{attribute addProperty BoxType "EK1122-0000-0018"}
{attribute addProperty Id "Beckhoff_EL73xxsub_EK1100EK1100_179A0949162"}
{attribute addProperty CRC "4226893576"}
{attribute addProperty SizeInBites "16"}
{attribute addProperty SizeInBytes "2"}
TYPE Beckhoff_EL73xxEK1122_FBF14708 EXTENDS EK1122_179A0949 :
STRUCT
	{attribute addProperty Name "Beckhoff_EL73xxsub_EK1100"}
	Beckhoff_EL73xxsub_EK1100 : EK1100_179A0949;
END_STRUCT
END_TYPE

(* stored: Version 1.2.0.0, ProductVersion 3.1.4024.9
   DUT Beckhoff_EL73xxEK1122_FBF14708: Id {0c4d4103-083b-4b4e-86fd-884bb9d9705f} *)
